Staubli VAL3: setErrorCode.pgx

program setErrorCode(num x_nAxisNum (dimensions=1), num& x_nErrorCode (dimensions=1))
  local num l_nAlarm
begin
  // This program returns the value of the current error
  //获取当前错误代码值
  x_nErrorCode=0
  //检查电机错误位是否被设置
  // Check if driveFault bit is set
  //  if diFault[x_nAxisNum]==true
  //    //硬件错误
  //    // Hardware alarm ?
  //    call chkHwAlarm(x_nAxisNum,x_nErrorCode)
  //    if x_nErrorCode==0
  //      // Software alarm ?
  //      call chkSwAlarm(x_nAxisNum,x_nErrorCode)
  //    endIf
  //    // Check alarm bits of status_remote register
  //  elseIf nAppV3Error[x_nAxisNum]==0
  //    call getRegisterVal(cst:nSTATUS_REMOTE,x_nAxisNum,x_nErrorCode)
  //  else
  //    // Check if Application error
  //    x_nErrorCode=nAppV3Error[x_nAxisNum]
  //  endIf
end
